VAR_GLOBAL
	g_IOCHostIP	: T_IPv4Addr := '127.0.0.1';
	g_udpSyslog	:	UDINT := 514;
	gMesgBuffer	:	ARRAY [0..cMesgArraySize] OF T_MaxString;
END_VAR
VAR_GLOBAL CONSTANT
	acsSubsystems	:	ARRAY [0..4] OF STRING := 
	['VACUUM', 'MPS', 'MOTION', 'FIELDBUS', '-'];
	cNILVALUE	:	STRING(1) := '-';
	cMesgArraySize : INT := 50;
END_VAR

(* stored: Version 1.1.0.1, ProductVersion 3.1.4018.5
   GVL GVL_Logger: Id {047a20cc-a785-4614-8465-ede098785b35} *)
